RESOURCE_TYPE _CoreSingle
  (* Standard: 61499-2 *)
  (* Version 0.1, 2017-00-22, hpea485, UOA *)
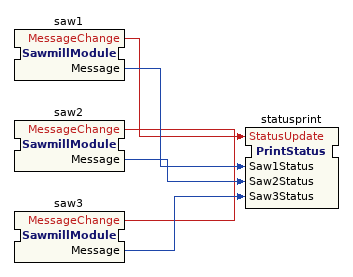
  FBS
    saw1 : SawmillModule;
    saw2 : SawmillModule;
    saw3 : SawmillModule;
    statusprint : PrintStatus;
  END_FBS
  EVENT_CONNECTIONS
    saw1.MessageChange TO statusprint.StatusUpdate;
    saw2.MessageChange TO statusprint.StatusUpdate;
    saw3.MessageChange TO statusprint.StatusUpdate;
  END_CONNECTIONS
  DATA_CONNECTIONS
    saw1.Message TO statusprint.Saw1Status;
    saw2.Message TO statusprint.Saw2Status;
    saw3.Message TO statusprint.Saw3Status;
  END_CONNECTIONS
END_RESOURCE_TYPE
